INTERFACE IPAFDosing EXTENDS IPAProcessFunction

END_INTERFACE

(* stored: Version 1.1.0.1, ProductVersion 3.1.4020.12
   Itf IPAFDosing: Id {381c707c-d678-481d-94e6-e89fdd5bb556} *)
